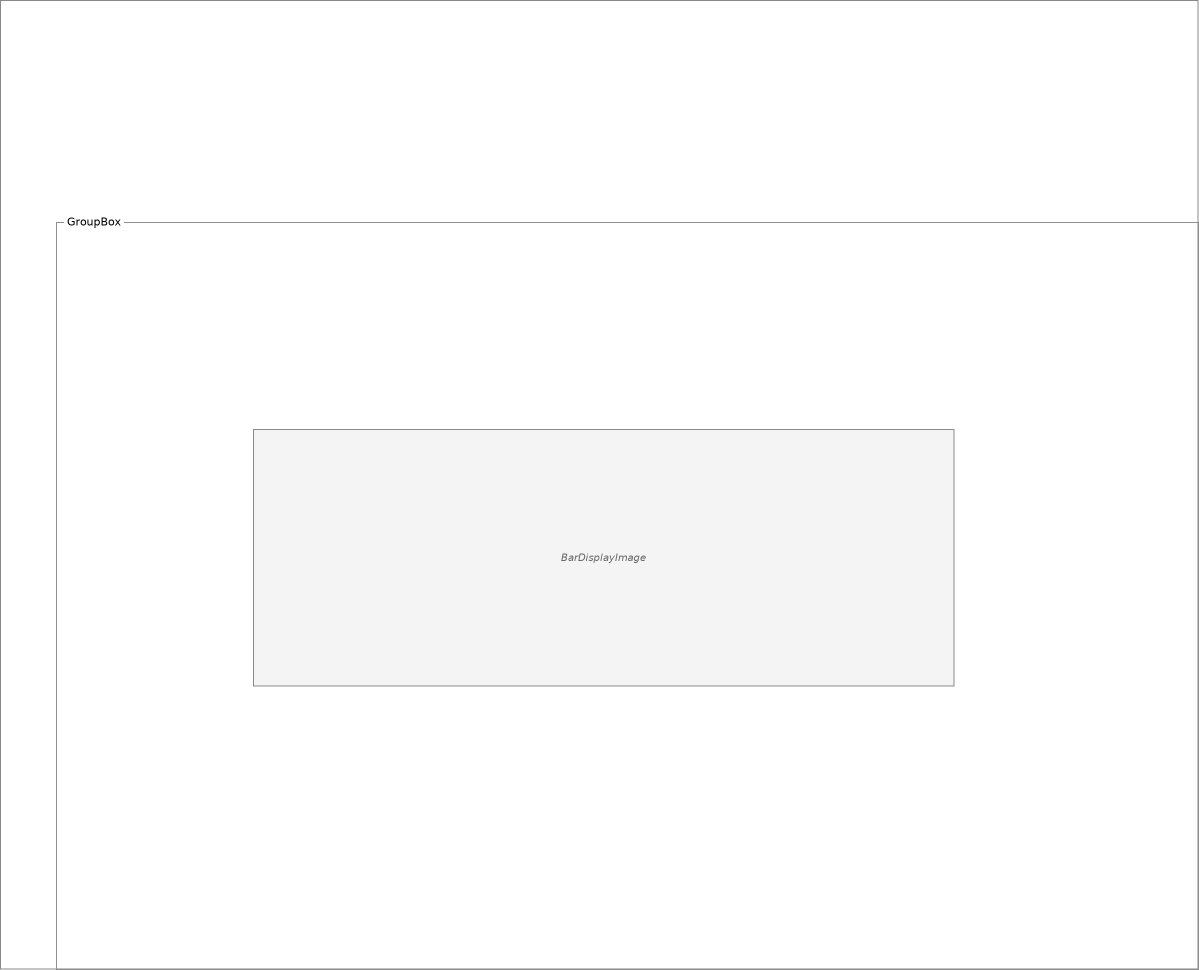
VISUALIZATION HMI_Crane  // 1199x970
    GroupBox (56,214 1143x756), "GroupBox"
        BarDisplayImage (197,215 701x257), value: G_MotionRef.fMotionGeneratorPos, style: BarDisplayImage-Gray, scale format: %.1f, scale 0..10
END_VISUALIZATION

(* stored: Version 1.1.0.1, ProductVersion 3.1.4024.12
   Visu HMI_Crane: Id {a8c570be-400d-4f7a-8a23-e8216c05248c} *)
